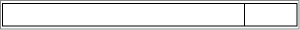
VISUALIZATION Vis_DigitalInput_2  // 300x30
VAR_IN_OUT
	stHMI_DigitalInput:stHMI_DigitalInput;
END_VAR
    Rectangle (2,3 243x23)
    Rectangle (244,3 53x23)
END_VISUALIZATION

(* stored: Version 1.1.0.1, ProductVersion 3.1.4024.11
   Visu Vis_DigitalInput_2: Id {680bbfb5-43b8-4aa8-bdd1-deedeff8cd8c} *)
